FUNCTION_BLOCK FB_HMIEMenu EXTENDS FB_BaseControlElement IMPLEMENTS ITF_HMIEMenu, ITF_HMIEMenu_HMI_Init
VAR
	arrButtons				: ARRAY [0..GVL_HMIEConstans.MAX_NUMBER_OF_BUTTON_IN_MENU] OF ITF_HMIEButton;
	iNumberOfButton			: INT := -1;	//ilosć przycisków w menu
	iActiveButton			: INT;	//numer aktywnego przycisku
	iActiveButtonPrev		: INT;
	bChangePage				: BOOL; //zmiana strony
END_VAR

METHOD PUBLIC AddButton : BOOL
VAR_INPUT
	fbButton			: ITF_HMIEButton;
END_VAR
IF (THIS^.iNumberOfButton + 1 <= GVL_HMIEConstans.MAX_NUMBER_OF_BUTTON_IN_MENU) THEN
	THIS^.iNumberOfButton := THIS^.iNumberOfButton + 1;
	THIS^.arrButtons [THIS^.iNumberOfButton] := fbButton;
	THIS^.arrButtons [THIS^.iNumberOfButton].SetEnable (bIN := TRUE);
	THIS^.arrButtons [THIS^.iNumberOfButton].SetVisible (bIN := TRUE);
	THIS^.AddComponent (itfComponent := fbButton);
	AddButton := TRUE;
ELSE
	AddButton := FALSE;
END_IF
END_METHOD

METHOD PUBLIC GetNumberOfActrivePreviewScreen : INT
VAR_INPUT
END_VAR
GetNumberOfActrivePreviewScreen := THIS^.iActiveButtonPrev;
END_METHOD

METHOD PUBLIC GetNumberOfActriveScreen : INT
VAR_INPUT
END_VAR
GetNumberOfActriveScreen := THIS^.iActiveButton;
END_METHOD

METHOD PUBLIC GetNumberOfAddedButton : INT
VAR_INPUT
END_VAR
GetNumberOfAddedButton := THIS^.iNumberOfButton;
END_METHOD

METHOD PUBLIC GetTitleOfActivePage : WSTRING
VAR_INPUT
END_VAR
//GetTitleOfActivePage := this^.arrButtons [this^.iActiveButton].GetName ();
END_METHOD

METHOD IsActiveButton : BOOL
VAR_INPUT
	iButton		: INT;	//numer przycisku
	bIN			: BOOL;
END_VAR
IsActiveButton	:= THIS^.arrButtons [iButton].IsActive ();
END_METHOD

METHOD PUBLIC IsChangePage : BOOL
VAR_INPUT
END_VAR
IsChangePage := THIS^.bChangePage;
END_METHOD

METHOD IsEnableButton : BOOL
VAR_INPUT
	iButton		: INT;	//numer przycisku
	bIN			: BOOL;
END_VAR
IsEnableButton	:= THIS^.arrButtons [iButton].IsEnable ();
END_METHOD

METHOD IsVisibleButton : BOOL
VAR_INPUT
	iButton		: INT;	//numer przycisku
	bIN			: BOOL;
END_VAR
IsVisibleButton	:= THIS^.arrButtons [iButton].IsVisible ();
END_METHOD

METHOD PUBLIC ResetChangePage
VAR_INPUT
END_VAR
THIS^.bChangePage := FALSE;
END_METHOD

METHOD SetActiveButton : BOOL
VAR_INPUT
	iButton		: INT;	//numer przycisku
	bIN			: BOOL;
END_VAR
THIS^.arrButtons [iButton].SetActive (bIN := bIN);
END_METHOD

METHOD SetEnableButton : BOOL
VAR_INPUT
	iButton		: INT;	//numer przycisku
	bIN			: BOOL;
END_VAR
THIS^.arrButtons [iButton].SetEnable (bIN := bIN);
END_METHOD

METHOD SetVisibleButton : BOOL
VAR_INPUT
	iButton		: INT;	//numer przycisku
	bIN			: BOOL;
END_VAR
THIS^.arrButtons [iButton].SetVisible (bIN := bIN);
END_METHOD

(*			
	RafalOS
	Rafał Osajda		11.11.2025		TC 4024.66
	testuje czy jest coś naciśnięte w menu i przełącza
*)
METHOD PUBLIC Testing : BOOL
VAR
	iI		: INT;
	iJ		: INT;
END_VAR
FOR iI := 0 TO THIS^.iNumberOfButton DO
	IF (THIS^.arrButtons [iI].IsPressed ()) THEN
		FOR iJ := 0 TO THIS^.iNumberOfButton DO 
			THIS^.arrButtons [iJ].SetActive (bIN := FALSE);
		END_FOR
		THIS^.arrButtons [iI].SetPressed (bIN := FALSE);
		THIS^.arrButtons [iI].SetActive (bIN := TRUE);
		THIS^.iActiveButtonPrev := THIS^.iActiveButton;
		THIS^.iActiveButton := iI;
		THIS^.bChangePage := TRUE;
	END_IF
END_FOR
END_METHOD

END_FUNCTION_BLOCK

(* stored: Version 1.1.0.1
   POU FB_HMIEMenu: Id {aca5b8d6-8bd3-4247-801c-4d7202167bd3}, SpecialFunc None
   Folder ITF_HMIEMenu: Id {4b3a4679-e153-0f1c-0cf6-c4b1dfee1813}
   Method AddButton: Id {84c5fa09-21a3-408e-a468-e17b66190995}
   Method GetNumberOfActrivePreviewScreen: Id {bc1974a1-9289-063d-1b9a-5c2077cdc82b}
   Method GetNumberOfActriveScreen: Id {98ddb291-5f6a-05ea-22f7-6340aae7623a}
   Method GetNumberOfAddedButton: Id {d4afd020-cb51-0d9c-3094-74d7a76ca847}
   Method GetTitleOfActivePage: Id {4dfec56d-8e66-0e98-2e07-c6efc333db3e}
   Method IsActiveButton: Id {b4d1a0ff-bd9d-0a66-1dc5-0550ed0d188d}
   Method IsChangePage: Id {8bd78c0c-f9d1-037d-04be-4e292db60507}
   Method IsEnableButton: Id {217e2c6a-563a-08bd-0fa4-1cc88765e86d}
   Method IsVisibleButton: Id {20df5edd-f349-000a-1620-91b9a13457e8}
   Method ResetChangePage: Id {2630c3ba-0ff9-0859-1451-9a6bf39714eb}
   Method SetActiveButton: Id {4a3f2cd9-b9dc-0e5a-20ae-b9e5849184e6}
   Method SetEnableButton: Id {09238708-59e8-0f4e-3df3-b9bd70508c9d}
   Method SetVisibleButton: Id {9b32dc56-5171-0eb1-09b1-fe51305e187e}
   Method Testing: Id {8201623d-ba65-073c-2675-52346bd25414} *)
